PROGRAM MAIN
VAR
	P_Axis_1_COMMAND AT%QD0:P_Axis_Tx;
	P_Axis_1_STATUS AT%ID0:P_Axis_Rx;
	
	P_Axis_2_COMMAND AT%QD3:P_Axis_Tx;
	P_Axis_2_STATUS AT%ID2:P_Axis_Rx;
	
	T_Axis_1_COMMAND AT%QD100:T_Axis_Tx;
	T_Axis_1_STATUS AT%ID100:T_Axis_Rx;
END_VAR

END_PROGRAM

(* stored: Version 1.1.0.1, ProductVersion 3.1.4024.12
   POU MAIN: Id {912dd12d-1b55-414e-be12-f9f02a64d7ff}, SpecialFunc None *)
